Fanuc KAREL source: kf00089.KL

-- PROVISIONAL review KL for V940-1; original PC SHA256 1e54331cb7a210a207c074f8b6123951f83ff4ff0c0cf6e6dde578b38c1eb419
-- Incomplete behavior may be omitted. Consult companion uncertainty JSON. Do not deploy.
PROGRAM KF00089
%NOLOCKGROUP
VAR
  I : INTEGER
  J : INTEGER
  X : REAL
  Y : REAL
  B : BOOLEAN
  C : BOOLEAN
  TXT : STRING[80]
  TXT2 : STRING[80]
  STATUS : INTEGER
-- UNRESOLVED_DECL AI type=002010
-- UNRESOLVED_DECL BI type=002010
-- UNRESOLVED_DECL P type=000102
-- UNRESOLVED_DECL JP type=000199
-- UNRESOLVED_DECL PF type=000101
-- UNRESOLVED_DECL V1 type=000013
-- UNRESOLVED_DECL V2 type=000013
BEGIN
  -- V9_ZERO_TABLE_METADATA_HINT layout=0001; no indexed target words; source/name/runtime held
  -- UNRESOLVED_PC offsets 5-32; opcodes 27,22,1C,76,7E,4A
  -- UNRESOLVED_PC offsets 37-41; opcodes 7F
END KF00089
